TYPE "Scanner_Write_Data"
VERSION : 0.1
   STRUCT
      Send_Data : Bool;
      Scanner_ID : Int;
      Scaner_Scan_Status : Int;
      Write_Int : Int;
      Error_Comment : String;
      Scan_Time : Date_And_Time;
   END_STRUCT;

END_TYPE

